// TIA Portal V19 export
FUNCTION_BLOCK "FAK_Updater_Type_PLen"   // FB127, LAD
TITLE = FAK UPDATER USING PART LENGTH / FAK UPDATER
// stored: Access Published, MemoryReserve 100, SetENOAutomatically false
   VAR_INPUT
      SystemEnable : Bool;
      MaterialCounter_Data : "MatCountData";
      Len : Struct
         ID : DInt;
         Val : LReal;
      END_STRUCT;
      PLen_Desired : LReal;
      Par { ExternalAccessible := 'False'; ExternalVisible := 'False'; ExternalWritable := 'False'} : Struct
         Enable : Bool;
         Apply_Enable : Bool;
         MaxWrongQty : UInt;
         Avg_ItemsQty : UInt;
         Avg_ErrTol : LReal;
         Tol_GOOD : LReal;
      END_STRUCT;
   END_VAR
   VAR_OUTPUT
      FAK_Apply : Bool;   // ApplyNewFAKRequired
      FAK_Value : LReal;
   END_VAR
   VAR
      HMI : Struct
         Button_INIT : Bool;
         Status_INIT_Done : Bool;
         Ststus_Operating : Bool;
         Status_FAK_Updater : Int;
         FAK_Calculated : LReal;
         PLen_Avg : LReal;
         Err_Avg : LReal;
         Buffer : Array[1..#BUFFER_ITEMS] of Struct
            Value : LReal;
            Err : LReal;
            Status : Int;
         END_STRUCT;
      END_STRUCT;
      FAK_ChangeReq : Bool;
      i : Int;
      Data : Struct
         Counter_Wrong : UInt;
         Counter_Good : UInt;
         LenSum : LReal;
         Err_AvgAbs { ExternalAccessible := 'False'; ExternalVisible := 'False'; ExternalWritable := 'False'} : LReal;
      END_STRUCT;
      PLen_Desired_Save : LReal;
      FAK_Save { S7_SetPoint := 'True'} : LReal;
      ID_Save : DInt;
      Aux : Struct
         StatusOperating_PE : Bool;
         StatusOperating_NE : Bool;
         HMI_ButtonINIT : Bool;
      END_STRUCT;
      TON_Init : TON_TIME;
   END_VAR
   VAR_TEMP
      PLen_Desiderd_IsChange : Bool;
      FAK_IsChange : Bool;
      Init : Bool;
      Init_Avg : Bool;
      New_Val : Bool;
   END_VAR
   VAR CONSTANT
      BUFFER_ITEMS : Int := 10;
      STATUS_PLEN_NULL : Int := 0;
      STATUS_PLEN_GOOD : Int := 2;
      STATUS_PLEN_WRONG : Int := 3;
      STATUS_FAK_UPDATER_WHITE : Int := 0;
      STATUS_FAK_UPDATER_GREEN : Int := 1;
      STATUS_FAK_UPDATER_YELLOW : Int := 2;
      STATUS_FAK_UPDATER_RED : Int := 3;
   END_VAR
   VAR_TEMP   // added for the SCL form of the ladder/FBD networks
      _w1 : Bool;
      _w2 : Bool;
      _w3 : Bool;
   END_VAR
BEGIN

REGION Network 1: Operating ON
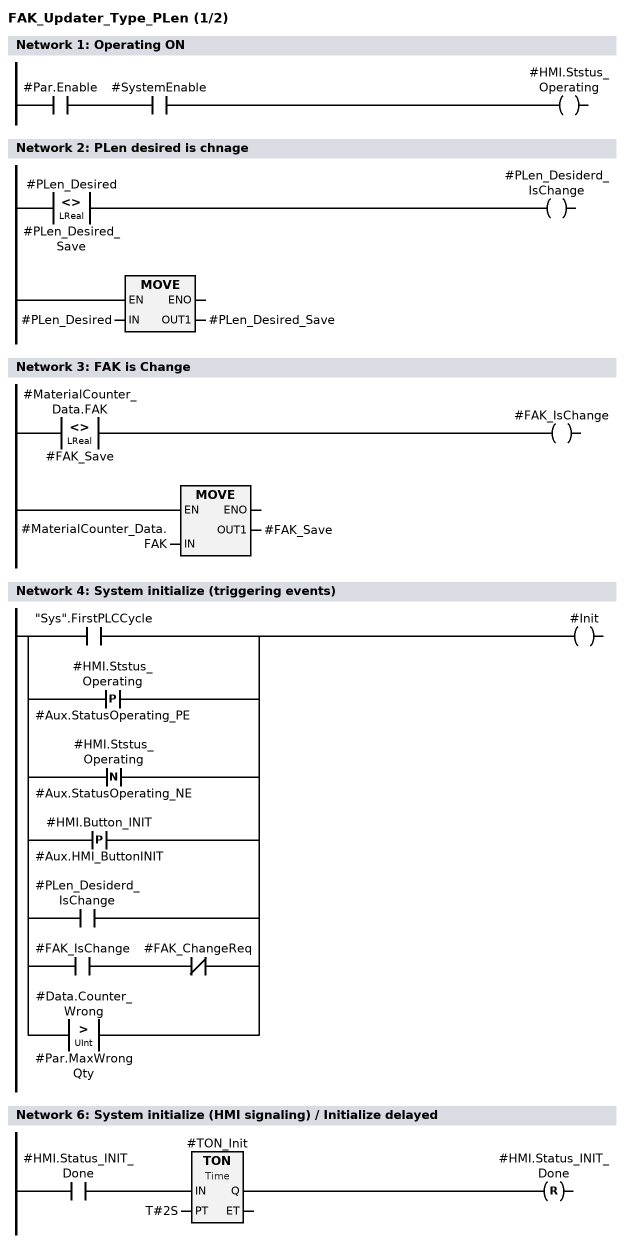
   RUNG wire#powerrail
      Contact( #Par.Enable )
      Contact( #SystemEnable )
      Coil( #HMI.Ststus_Operating )
   END_RUNG
   // the same network as SCL:
   #HMI.Ststus_Operating := #Par.Enable AND #SystemEnable;
END_REGION

REGION Network 2: PLen desired is chnage
   RUNG wire#powerrail
      { S7_Templates := "SrcType := LReal" } NE_Contact(in1 := #PLen_Desired, in2 := #PLen_Desired_Save)
      Coil( #PLen_Desiderd_IsChange )
   END_RUNG
   RUNG wire#powerrail
      { S7_GenerateENO := "TRUE" } Move(in := #PLen_Desired, out1 => #PLen_Desired_Save)
   END_RUNG
   // the same network as SCL:
   #PLen_Desiderd_IsChange := #PLen_Desired <> #PLen_Desired_Save;
   #PLen_Desired_Save := #PLen_Desired;
END_REGION

REGION Network 3: FAK is Change
   RUNG wire#powerrail
      { S7_Templates := "SrcType := LReal" } NE_Contact(in1 := #MaterialCounter_Data.FAK, in2 := #FAK_Save)
      Coil( #FAK_IsChange )
   END_RUNG
   RUNG wire#powerrail
      { S7_GenerateENO := "TRUE" } Move(in := #MaterialCounter_Data.FAK, out1 => #FAK_Save)
   END_RUNG
   // the same network as SCL:
   #FAK_IsChange := #MaterialCounter_Data.FAK <> #FAK_Save;
   #FAK_Save := #MaterialCounter_Data.FAK;
END_REGION

REGION Network 4: System initialize (triggering events)
   RUNG wire#powerrail
      Contact( "Sys".FirstPLCCycle )
      wire#w1
      Coil( #Init )
   END_RUNG
   RUNG wire#powerrail
      P_Contact(operand := #HMI.Ststus_Operating, bit := #Aux.StatusOperating_PE)
   END_RUNG wire#w1
   RUNG wire#powerrail
      N_Contact(operand := #HMI.Ststus_Operating, bit := #Aux.StatusOperating_NE)
   END_RUNG wire#w1
   RUNG wire#powerrail
      P_Contact(operand := #HMI.Button_INIT, bit := #Aux.HMI_ButtonINIT)
   END_RUNG wire#w1
   RUNG wire#powerrail
      Contact( #PLen_Desiderd_IsChange )
   END_RUNG wire#w1
   RUNG wire#powerrail
      Contact( #FAK_IsChange )
      I_Contact( #FAK_ChangeReq )
   END_RUNG wire#w1
   RUNG wire#powerrail
      { S7_Templates := "SrcType := UInt" } GT_Contact(in1 := #Data.Counter_Wrong, in2 := #Par.MaxWrongQty)
   END_RUNG wire#w1
   // the same network as SCL:
   #_w1 := #HMI.Ststus_Operating AND NOT #Aux.StatusOperating_PE;   // rising edge of #HMI.Ststus_Operating
   #Aux.StatusOperating_PE := #HMI.Ststus_Operating;
   #_w2 := NOT #HMI.Ststus_Operating AND #Aux.StatusOperating_NE;   // falling edge of #HMI.Ststus_Operating
   #Aux.StatusOperating_NE := #HMI.Ststus_Operating;
   #_w3 := #HMI.Button_INIT AND NOT #Aux.HMI_ButtonINIT;   // rising edge of #HMI.Button_INIT
   #Aux.HMI_ButtonINIT := #HMI.Button_INIT;
   #Init := "Sys".FirstPLCCycle OR #_w1 OR #_w2 OR #_w3 OR #PLen_Desiderd_IsChange OR (#FAK_IsChange AND NOT #FAK_ChangeReq) OR (#Data.Counter_Wrong > #Par.MaxWrongQty);
END_REGION

REGION Network 5 (SCL): System initialize (execution)
   IF #Init THEN

       #HMI.Status_INIT_Done := TRUE;
       #FAK_ChangeReq := FALSE;

       #ID_Save := #Len.ID;


       #Data.Counter_Wrong := 0;
       #Data.Counter_Good := 0;
       #Data.LenSum := 0;
       #Data.Err_AvgAbs := 0;


       #HMI.FAK_Calculated :=  #MaterialCounter_Data.FAK;
       #HMI.Err_Avg :=  0.0;
       #HMI.PLen_Avg := #PLen_Desired;



       #HMI.Status_FAK_Updater := #STATUS_FAK_UPDATER_WHITE;


       FOR #i := 1 TO #BUFFER_ITEMS DO

           #HMI.Buffer[#i].Value := 0.0;
           #HMI.Buffer[#i].Err := 0.0;
           #HMI.Buffer[#i].Status := #STATUS_PLEN_NULL;

       END_FOR;



   END_IF;
END_REGION

REGION Network 6: System initialize (HMI signaling) / Initialize delayed
   RUNG wire#powerrail
      Contact( #HMI.Status_INIT_Done )
      { S7_Templates := "time_type := Time" } #TON_Init.TON(pt := T#2S, et =>)
      R_Coil( #HMI.Status_INIT_Done )
   END_RUNG
   // the same network as SCL:
   #TON_Init(IN := #HMI.Status_INIT_Done, PT := T#2S);   // TON
   IF #TON_Init.Q THEN #HMI.Status_INIT_Done := FALSE; END_IF;
END_REGION

REGION Network 7: New item to load
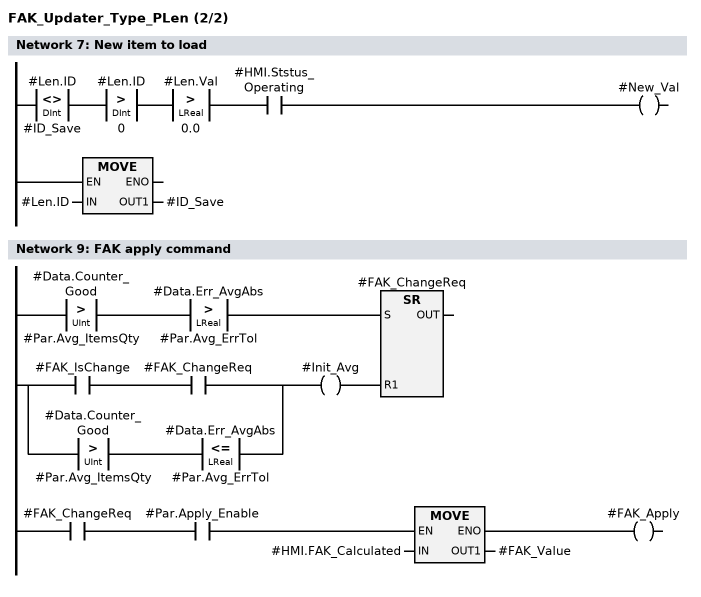
   RUNG wire#powerrail
      { S7_Templates := "SrcType := DInt" } NE_Contact(in1 := #Len.ID, in2 := #ID_Save)
      { S7_Templates := "SrcType := DInt" } GT_Contact(in1 := #Len.ID, in2 := 0)
      { S7_Templates := "SrcType := LReal" } GT_Contact(in1 := #Len.Val, in2 := 0.0)
      Contact( #HMI.Ststus_Operating )
      Coil( #New_Val )
   END_RUNG
   RUNG wire#powerrail
      Move(in := #Len.ID, out1 => #ID_Save)
   END_RUNG
   // the same network as SCL:
   #New_Val := (#Len.ID <> #ID_Save) AND (#Len.ID > 0) AND (#Len.Val > 0.0) AND #HMI.Ststus_Operating;
   #ID_Save := #Len.ID;
END_REGION

REGION Network 8 (SCL): Buffer TP - Push item
   IF #New_Val THEN


       #i := #BUFFER_ITEMS;

       WHILE #i >= 2 DO

           #HMI.Buffer[#i] := #HMI.Buffer[#i - 1];

           #i -= 1;

       END_WHILE;


       #HMI.Buffer[1].Value := #Len.Val;
       #HMI.Buffer[1].Err := #Len.Val - #PLen_Desired;



       IF ABS(#HMI.Buffer[1].Err) <= #Par.Tol_GOOD THEN

           #HMI.Buffer[1].Status := #STATUS_PLEN_GOOD;

           #Data.Counter_Good += 1;

           #Data.LenSum := #Data.LenSum + #HMI.Buffer[1].Value;


           #HMI.PLen_Avg := #Data.LenSum / #Data.Counter_Good ;

           #HMI.Err_Avg :=  #HMI.PLen_Avg - #PLen_Desired;

           #Data.Err_AvgAbs := ABS(#HMI.Err_Avg);


           #HMI.FAK_Calculated := #PLen_Desired / #HMI.PLen_Avg * #MaterialCounter_Data.FAK;


           IF #HMI.Err_Avg < (#Par.Avg_ErrTol / 2.0) THEN

               #HMI.Status_FAK_Updater := #STATUS_FAK_UPDATER_GREEN; // Verde;

           ELSIF  #HMI.Err_Avg > #Par.Avg_ErrTol THEN

               #HMI.Status_FAK_Updater := #STATUS_FAK_UPDATER_RED; // Rosso;

           ELSE
               #HMI.Status_FAK_Updater := #STATUS_FAK_UPDATER_YELLOW; // Giallo;

           END_IF;


       ELSE

           #Data.Counter_Wrong += 1;

           #HMI.Buffer[1].Status := #STATUS_PLEN_WRONG;


       END_IF;


   END_IF;
END_REGION

REGION Network 9: FAK apply command
   RUNG wire#powerrail
      { S7_Templates := "SrcType := UInt" } GT_Contact(in1 := #Data.Counter_Good, in2 := #Par.Avg_ItemsQty)
      { S7_Templates := "SrcType := LReal" } GT_Contact(in1 := #Data.Err_AvgAbs, in2 := #Par.Avg_ErrTol)
      S_SR(operand := #FAK_ChangeReq, r1 := wire#w2)
   END_RUNG
   RUNG wire#powerrail
      Contact( #FAK_IsChange )
      Contact( #FAK_ChangeReq )
      wire#w1
      Coil( #Init_Avg )
   END_RUNG wire#w2
   RUNG wire#powerrail
      { S7_Templates := "SrcType := UInt" } GT_Contact(in1 := #Data.Counter_Good, in2 := #Par.Avg_ItemsQty)
      { S7_Templates := "SrcType := LReal" } LE_Contact(in1 := #Data.Err_AvgAbs, in2 := #Par.Avg_ErrTol)
   END_RUNG wire#w1
   RUNG wire#powerrail
      Contact( #FAK_ChangeReq )
      Contact( #Par.Apply_Enable )
      { S7_GenerateENO := "TRUE" } Move(in := #HMI.FAK_Calculated, out1 => #FAK_Value)
      Coil( #FAK_Apply )
   END_RUNG
   // the same network as SCL:
   // ENO of a box is taken as its EN; it also drops when the box reports an error
   #Init_Avg := (#FAK_IsChange AND #FAK_ChangeReq) OR ((#Data.Counter_Good > #Par.Avg_ItemsQty) AND (#Data.Err_AvgAbs <= #Par.Avg_ErrTol));
   IF (#Data.Counter_Good > #Par.Avg_ItemsQty) AND (#Data.Err_AvgAbs > #Par.Avg_ErrTol) THEN
       #FAK_ChangeReq := TRUE;   // SR flip-flop
   END_IF;
   IF #Init_Avg THEN #FAK_ChangeReq := FALSE; END_IF;
   #_w1 := #FAK_ChangeReq AND #Par.Apply_Enable;
   IF #_w1 THEN #FAK_Value := #HMI.FAK_Calculated; END_IF;
   #FAK_Apply := #_w1;
END_REGION

REGION Network 10 (SCL): Init Average
   IF #Init_Avg THEN


       #Data.Counter_Wrong := 0;
       #Data.Counter_Good := 0;
       #Data.LenSum := 0;
       #Data.Err_AvgAbs := 0;


       #HMI.FAK_Calculated :=  #MaterialCounter_Data.FAK;
       #HMI.Err_Avg :=  0.0;
       #HMI.PLen_Avg := #PLen_Desired;



       #HMI.Status_FAK_Updater := #STATUS_FAK_UPDATER_WHITE;



   END_IF;
END_REGION

REGION Network 11: >
END_REGION

REGION Network 12: >
END_REGION

REGION Network 13: >
END_REGION
END_FUNCTION_BLOCK
